Staubli VAL3: changeSpeed.pgx

program changeSpeed(num x_nType, num x_nIndex)
  local string l_sMessage[2]
  local num l_nActual
  local num l_nOldValue
  local num l_nSize
  local num i
begin
  //
  // change all the speed
  //
  switch x_nType
    case 0
      // APPROACH
      call language2:message(l_sMessage,0)
      call language2:message(l_sMessage[1],2)
      l_nActual=l_nOldValue=pEditPoint.nSpeedApproach
      call use:insertDialog(l_sMessage+" "+l_sMessage[1],pEditPoint.nSpeedApproach,1,6000)
    break
    case 1
      // DEPART
      call language2:message(l_sMessage,1)
      call language2:message(l_sMessage[1],2)
      l_nActual=l_nOldValue=pEditPoint.nSpeedDepart
      call use:insertDialog(l_sMessage+" "+l_sMessage[1],pEditPoint.nSpeedDepart,1,6000)
    break
    case 2
      // NORMAL SPEED
      call language:message(l_sMessage,161)
      if pEditPoint.tData[x_nIndex].tSuper.moveType==0
        l_nActual=l_nOldValue=pEditPoint.tData[x_nIndex].tSuper.nom_speed.vel
        call use:insertDialog(l_sMessage,l_nActual,1,400)
      else
        if pEditPoint.tData[x_nIndex].tSuper.moveType==1
          l_nActual=l_nOldValue=pEditPoint.tData[x_nIndex].tSuper.nom_speed.tvel
          call use:insertDialog(l_sMessage,l_nActual,1,6000)
        endIf
      endIf
    break
  endSwitch
  // set all the speed
  if l_nActual!=l_nOldValue and x_nType==2
    // normal speed, 2
    call getSizeItem(false,l_nSize)
    for i=0 to (l_nSize-1)
      if (pEditPoint.tData[i].tSuper.moveType==0)and(l_nOldValue==pEditPoint.tData[i].tSuper.nom_speed.vel)
        pEditPoint.tData[i].tSuper.nom_speed.vel=l_nActual
      else
        if (pEditPoint.tData[i].tSuper.moveType==1)and(l_nOldValue==pEditPoint.tData[i].tSuper.nom_speed.tvel)
          pEditPoint.tData[i].tSuper.nom_speed.tvel=l_nActual
        endIf
      endIf
    endFor
  endIf
  // to be saved
  bToSave=true
end
